INTERFACE I_Request EXTENDS I_Disposable

PROPERTY PUBLIC CreatedTimestamp : I_Timestamp
GET
END_GET
END_PROPERTY

PROPERTY PUBLIC Header : I_Header
GET
END_GET
END_PROPERTY

PROPERTY PUBLIC PayloadAddress : POINTER TO STRING
GET
END_GET
END_PROPERTY

PROPERTY PUBLIC PayloadSizeInBytes : UDINT
GET
END_GET
END_PROPERTY

END_INTERFACE

(* stored: Version 1.1.0.1, ProductVersion 3.1.4024.12
   Itf I_Request: Id {bbe5c3e3-282c-0b95-03ec-2f91b02573a7}
   Property CreatedTimestamp: Id {a125f5ac-6b94-06e9-28a6-40f783f1f01c}
   Get Get: Id {6d623bd0-919d-0543-0060-77b4100af55f}
   Property Header: Id {f7024f20-5c72-06e1-3653-6fab0f8ea0c1}
   Get Get: Id {171c1529-f942-0beb-12d2-6c9cba2dfebe}
   Property PayloadAddress: Id {a1e27b07-c91a-0410-3f66-72405e0766c8}
   Get Get: Id {6e2621cd-1042-0f01-1b9d-20f7bb99f879}
   Property PayloadSizeInBytes: Id {52dd94d9-0ec1-0930-305a-d23eec5f6209}
   Get Get: Id {2bd70307-aff7-0dba-1e42-064e536403cd} *)
